PROGRAM MAIN
VAR
END_VAR

EscreverDB();
LerDB();

END_PROGRAM

(* stored: Version 1.1.0.1
   POU MAIN: Id {59fead0d-6c10-4da3-a54a-c1a59097b339}, SpecialFunc None *)
